(* PLC project Generated.project, CODESYS CODESYS V3.5 SP19 Patch 1 *)
(* stored: creationDateTime 2026-07-30T14:51:12.632763, modificationDateTime 2026-07-30T14:51:12.632763 *)

(* ═══════════════════════════════════════════════════════════════ 🚦 ST_ModesState — États et diagnostics IHM des modes de marche ═══════════════════════════════════════════════════════════════ *)
TYPE ST_ModesState : STRUCT
  CurrentMode : E_Mode;  (* 🎚️ Mode de marche actuellement actif *)
  PowerContactorEngaged : BOOL;  (* 🛡️ État de la chaîne d'arrêt d'urgence *)
  AnyFaultActive : BOOL;  (* 🔴 REX 2026-07-07 : au moins un défaut/alarme actif dans le domaine *)
  PowerCutOffActive : BOOL;  (* 🧨 REX 2026-07-07 : au moins un Méca A/B/C (FB_Safety_Winch) ou *)
  EmergencyChainOk : BOOL;  (* 🔗 Boucle AU saine (coup-de-poing relâchés + pas de PowerCutOff PLC actif) *)
  PowerContactorOk : BOOL;  (* 🔌 Contacteur de puissance confirmé engagé (miroir PowerContactorEngaged) *)
  EmergencyArmable : BOOL;  (* 🟢 Réarmement possible maintenant (chaîne saine, ni séquence ni verrouillage en cours, *)
  EmergencyArmingBusy : BOOL;  (* ⏳ Auto-test A/B, pulse, confirmation OU verrouillage 5s en cours — nouvelle demande ignorée *)
  RedundancyTestFailed : BOOL;  (* 🔴 Canal A ou B non fonctionnel détecté à l'auto-test — bloque tout réarmement (front Reset requis) *)
  EmergencyArmingFailed : BOOL;  (* 🔴 Impulsion envoyée mais contacteur puissance jamais confirmé sous 2s (front Reset + contacteur confirmé requis) *)
END_STRUCT;
END_TYPE

(* values of E_Mode: DISABLE: Mode Désactivé / Veille de sécurité (sorties bloquées); MAINT_N1: Manuel Niveau 1 : Pilotage unitaire avec toutes sécurités actives; MAINT_N2: Manuel Niveau 2 : Pilotage dégradé (droits étendus + bypasses autorisés); SEMI_AUTO: Mode Semi-Automatique (séquenceur automatique) *)

{attribute 'qualified_only'}
{attribute 'strict'}
TYPE E_Mode : (DISABLE := 0, MAINT_N1 := 1, MAINT_N2 := 2, SEMI_AUTO := 3);
END_TYPE
